PROGRAM MAIN
VAR
	_test:Test;
	_running:BOOL;
END_VAR

_test();
_running := _test.Running;

END_PROGRAM

(* stored: Version 1.1.0.1, ProductVersion 3.1.4024.2
   POU MAIN: Id {972b3bb0-0ef7-4b5c-929a-ef97236f553a}, SpecialFunc None *)
